DATA_BLOCK "DB_maXYmosNC1"
{ S7_Optimized_Access := 'FALSE' }
VERSION : 0.1
NON_RETAIN
"KistlerPresser _FB"

BEGIN

END_DATA_BLOCK

